// SIMATIC S7-200 project (STEP 7-Micro/WIN), CPU 221 REL 01.10

ORGANIZATION_BLOCK PRINCIPAL:OB1
TITLE=Arranque con retardo - SET con retardo  /  JEVG
BEGIN
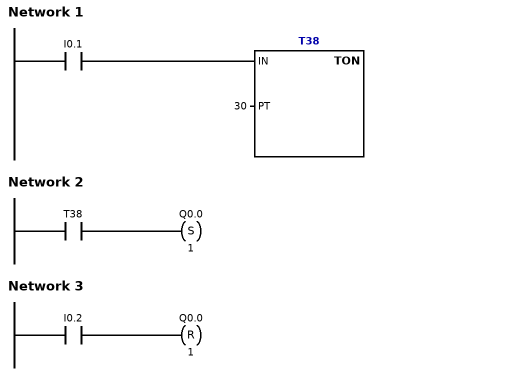
Network 1
// (network saved uncompiled; LAD cells follow)
// row 0: c0 -| |- I0.1  c1 --  c2 [TON T38 IN:=power@row0, PT:=30]
// row 1: c2 [box]
Network 2
LD     T38
S      Q0.0, 1
Network 3
LD     I0.2
R      Q0.0, 1
END_ORGANIZATION_BLOCK
